{attribute 'GeneratedUsingTerminal: EL6201-0000-0017'}
{attribute addProperty BoxType "EL6201-0000-0017"}
{attribute addProperty Id "Slave_18A_DI0BOOL1Slave_18A_DI1BOOL1Slave_18A_DI2BOOL1Slave_18A_DI3BOOL1Slave_18B_DI0BOOL1Slave_18B_DI1BOOL1Slave_18B_DI2BOOL1Slave_18B_DI3BOOL1"}
{attribute addProperty CRC "2280930463"}
{attribute addProperty Size "8"}
TYPE Slave_18_Inputs_87F43C9F :
STRUCT
	{attribute addProperty Name "Slave_18A_DI0"}
	Slave_18A_DI0 : BOOL;
	{attribute addProperty Name "Slave_18A_DI1"}
	Slave_18A_DI1 : BOOL;
	{attribute addProperty Name "Slave_18A_DI2"}
	Slave_18A_DI2 : BOOL;
	{attribute addProperty Name "Slave_18A_DI3"}
	Slave_18A_DI3 : BOOL;
	{attribute addProperty Name "Slave_18B_DI0"}
	Slave_18B_DI0 : BOOL;
	{attribute addProperty Name "Slave_18B_DI1"}
	Slave_18B_DI1 : BOOL;
	{attribute addProperty Name "Slave_18B_DI2"}
	Slave_18B_DI2 : BOOL;
	{attribute addProperty Name "Slave_18B_DI3"}
	Slave_18B_DI3 : BOOL;
END_STRUCT
END_TYPE

(* stored: Version 1.2.0.0, ProductVersion 3.1.4024.9
   DUT Slave_18_Inputs_87F43C9F: Id {784f1546-3a3a-452c-b7c7-b0fe648326ec} *)
